FUNCTION_BLOCK Test_TStreamAdd_Read_DINT EXTENDS T_UnitTestBase
VAR
    Stream  : T_Stream(StreamLength := 2);
    ArgType : E_ArgTypeId := E_ArgTypeId.Type_DINT;
END_VAR

Stream.Init(2);

// add a DINT...
Stream.SetNextArgTypeId(ArgType);
Stream.Add_DINT(12345678);

Stream.SetReadPosition(0);

// check next arg type is correct...
Assertion.AssertEquals_INT(Expected     := ArgType,
                           Actual       := Stream.GetNextArgTypeId(),
                           VariableName := 'Stream.GetNextArgTypeId()');

// check next value...	
Assertion.AssertEquals_DINT(Expected     := 12345678,
                            Actual       := Stream.Read_DINT(),
                            VariableName := 'Stream.Read_DINT()');

// check we are at the end of the stream..							
Assertion.AssertEquals_UDINT(Expected     := Stream.StreamLength,
                             Actual       := Stream.ReadPosition,
                             VariableName := 'Stream.ReadPosition');

TestFinished();

END_FUNCTION_BLOCK

(* stored: Version 1.1.0.1, ProductVersion 3.1.4024.9
   POU Test_TStreamAdd_Read_DINT: Id {41b01fdf-2f91-4c50-838b-71907799f62d}, SpecialFunc None *)
